(* PLC project Unnamed, Unknown Unnamed 1 *)
(* stored: creationDateTime 2013-01-29T14:01:00, modificationDateTime 2013-02-26T15:59:13 *)

FUNCTION_BLOCK GETVERSIONSTRING
  VAR_OUTPUT
    VERSION : STRING;
  END_VAR

{{
 #define STRINGify(x) __STRING_LITERAL(sizeof(#x),#x)
 STRING TMP = STRINGify(PLC_VERSION_STRING);
 SetFbVar(VERSION, TMP);
 #undef STRINGify
}}

          
END_FUNCTION_BLOCK
